(*			
	RafalOS
	Rafał Osajda		20.11.2025		TC 4024.66
	Moduł przygotowania danych dla Okna zmiany trybu we wszystkich trybach
*)
FUNCTION_BLOCK FB_MCHMIPrepareDataForScreen_04_XX EXTENDS FB_MCHMIPrepareDataForScreen IMPLEMENTS ITF_MCHMIPrepareDataForScreen
VAR
	itfMachineControlHMI	: ITF_MCHMIMachineControl_HMI_PrepScr_04_XX;
	refstData				: REFERENCE TO ST_MCHMIPrepareScreen_04_XX;
END_VAR

(*			
	RafalOS
	Rafał Osajda		19.11.2025		TC 4024.66
	Czyści danych przy zmienia ramki po poprzedniej ramce
*)
METHOD PUBLIC ClearAfterScreen : BOOL
VAR_INPUT
END_VAR
SUPER^.ClearAfterScreen ();
END_METHOD

METHOD PUBLIC LinkDataHMI_04_XX : BOOL
VAR_INPUT
	refstData				: REFERENCE TO ST_MCHMIPrepareScreen_04_XX;
END_VAR
THIS^.refstData REF= refstData;
END_METHOD

METHOD PUBLIC LinkMachineControlHMI : BOOL
VAR_INPUT
	fbMachineControlHMI	: ITF_MCHMIMachineControl_HMI_PrepScr_04_XX;
END_VAR
this^.itfMachineControlHMI := fbMachineControlHMI;
END_METHOD

(*			
	RafalOS
	Rafał Osajda		14.11.2025		TC 4024.66
	Metoda przygotowywania danych dla HMI 
	W niej odbywa się odpytywanie właściego elementu przez łącznik
*)
METHOD PUBLIC PrepareDataForHMI : BOOL
VAR_INST
	etmpMode					: E_BaseMachineMode := E_BaseMachineMode.NotAllowed;
END_VAR
VAR
	iJ							: INT;
	iActiveMode					: E_BaseMachineMode;
	etmpCmdChangeMode			: E_SaMCommandChangeMode;
END_VAR
THIS^.refstData.wsActualMode := THIS^.GetTextFromLabelForActiveLocation (THIS^.itfMachineControlHMI.GetActiveModeName ());
THIS^.refstData.eActualMode := THIS^.itfMachineControlHMI.GetActiveMode ();


	(*	Przygotowanie ifnormacji dla zmiany trybu	*)

IF (THIS^.refstHMICommonData.bChangePage OR etmpMode <> THIS^.refstData.eActualMode) THEN
	etmpMode := THIS^.refstData.eActualMode;
	THIS^.refstData.iNumberModeToDisplay := 0;
	iActiveMode := THIS^.itfMachineControlHMI.GetActiveMode ();
	FOR iJ := 1 TO GVL_SaMConstans.NUMBER_OF_MODES DO
		IF (THIS^.itfMachineControlHMI.IsModeEnabled (iMode := iJ) AND iJ <> iActiveMode) THEN
			THIS^.refstData.arrNamesOfMode [THIS^.refstData.iNumberModeToDisplay].wsDescription := 
				THIS^.GetTextFromLabelForActiveLocation (stLabel := THIS^.itfMachineControlHMI.GetModeName (iMode := iJ));
			THIS^.refstData.arrNamesOfMode [THIS^.refstData.iNumberModeToDisplay].iNumber := iJ;
			THIS^.refstData.iNumberModeToDisplay := THIS^.refstData.iNumberModeToDisplay + 1;
			THIS^.refstData.iSelectedMode := -1;
		END_IF
	END_FOR
END_IF
IF (THIS^.refstData.bChangeMode AND THIS^.refstData.bSelectedRow) THEN
	THIS^.refstData.bChangeMode := FALSE;
	//polecenie zmiany trybu 
	CASE THIS^.refstData.arrNamesOfMode [THIS^.refstData.iSelectedMode].iNumber OF
	E_SaMCommandChangeMode.Production : etmpCmdChangeMode := E_SaMCommandChangeMode.Production;
	E_SaMCommandChangeMode.Maintenance : etmpCmdChangeMode := E_SaMCommandChangeMode.Maintenance;
	E_SaMCommandChangeMode.Manual : etmpCmdChangeMode := E_SaMCommandChangeMode.Manual;
	E_SaMCommandChangeMode.Washing : etmpCmdChangeMode := E_SaMCommandChangeMode.Washing;
	E_SaMCommandChangeMode.Diagnostisc : etmpCmdChangeMode := E_SaMCommandChangeMode.Diagnostisc;
	END_CASE
	THIS^.itfMachineControlHMI.SetCmdChangeMode (eCmdNumber := etmpCmdChangeMode);
	THIS^.refstData.iSelectedMode := -1;
END_IF



SUPER^.PrepareDataForHMI ();
END_METHOD

(*			
	RafalOS
	Rafał Osajda		19.11.2025		TC 4024.66
	Przygotowanie ramki pood tamke do wyświetlenia - tylko przygotowanie a nie przygotowanie danych do wyświetlenia
*)
METHOD PUBLIC PrepareForScreen : BOOL
VAR_INPUT
END_VAR
SUPER^.PrepareForScreen ();
END_METHOD

END_FUNCTION_BLOCK

(* stored: Version 1.1.0.1
   POU FB_MCHMIPrepareDataForScreen_04_XX: Id {6e4dfaff-27c8-0025-119a-a34cf39f28f4}, SpecialFunc None
   Folder ITF_PDFS: Id {66ea2dcc-5128-071a-252d-f1f6604cbb90}
   Method ClearAfterScreen: Id {8287c1d6-fd3c-0f0a-0fd5-127913c425ee}
   Method LinkDataHMI_04_XX: Id {2e53909c-f49d-097b-3748-36ac1b2bd0b8}
   Method LinkMachineControlHMI: Id {081b03c4-328d-0073-21e2-a1ffff3db083}
   Method PrepareDataForHMI: Id {f50cac7c-a5ce-09f1-11e2-97991cebb006}
   Method PrepareForScreen: Id {b3c05c97-1dee-05a6-050f-2577330ebeb3} *)
